{attribute 'no_explicit_call' := 'do not call this POU directly'} 
FUNCTION_BLOCK FB_LoggerProxy IMPLEMENTS I_Logger
VAR_INPUT
END_VAR
VAR_OUTPUT
END_VAR
VAR
	pHead:				POINTER TO ST_LoggerNode;
END_VAR

//FB_Exit muss explizit implementiert werden. Wenn es eine Implementierung gibt, dann wird 
//die Methode aufgerufen, bevor die Steuerung den Code der Funktionsbaustein-Instanz entfernt
//(impliziter Aufruf. Der Rückgabewert wird nicht ausgewertet.
METHOD FB_Exit: BOOL
VAR_INPUT    
bInCopyCode: BOOL;  // TRUE: Die Exit-Methode wird aufgerufen, um die Instanz zu verlassen, die hinterher kopiert wird Online-Change).  
END_VAR
M_Clear();
END_METHOD

METHOD M_Attach : BOOL
VAR_INPUT
    iLogger : I_Logger;
END_VAR
VAR
    pCurrent : POINTER TO ST_LoggerNode;
END_VAR
// invalid input
IF iLogger = 0 THEN
    M_Attach := FALSE;
    RETURN;
END_IF

// first node
IF pHead = 0 THEN
    pHead := __NEW(ST_LoggerNode);
    IF pHead = 0 THEN
        RETURN;
    END_IF
    pHead^.iLogger := iLogger;
    pHead^.pNext := 0;
    M_Attach := TRUE;
    RETURN;
END_IF

// traverse list to check duplicates and reach last node
pCurrent := pHead;
WHILE pCurrent^.pNext <> 0 DO
    IF pCurrent^.iLogger = iLogger THEN
        M_Attach := FALSE; // already attached
        RETURN;
    END_IF
    pCurrent := pCurrent^.pNext;
END_WHILE

// check last node for duplicate
IF pCurrent^.iLogger = iLogger THEN
    RETURN;
END_IF

pCurrent^.pNext:= __NEW(ST_LoggerNode);
IF pCurrent^.pNext = 0 THEN
    RETURN;
END_IF
pCurrent^:= pCurrent^.pNext^;

pCurrent^.iLogger:= iLogger;
pCurrent^.pNext := 0;

M_Attach := TRUE;
END_METHOD

METHOD PUBLIC M_Clear : BOOL
VAR_INPUT
END_VAR
VAR
    pCurrent : POINTER TO ST_LoggerNode;
    pNext    : POINTER TO ST_LoggerNode;
END_VAR
pCurrent := pHead;

WHILE pCurrent <> 0 DO
    pNext := pCurrent^.pNext; // save next pointer
    __DELETE(pCurrent);       // free current node
    pCurrent := pNext;        // move to next node
END_WHILE

pHead := 0;                   // reset head
M_Clear := TRUE;
END_METHOD

METHOD M_Detach : BOOL
VAR_INPUT
	iLogger:			I_Logger;
END_VAR
VAR
    pCurrent : POINTER TO ST_LoggerNode;
    pPrev : POINTER TO ST_LoggerNode;
END_VAR
// invalid input
IF iLogger = 0 THEN
    RETURN;
END_IF

pCurrent := pHead;
pPrev := 0;
WHILE pCurrent <> 0 DO
    IF pCurrent^.iLogger = iLogger THEN
        IF pPrev = 0 THEN
            pHead := pCurrent^.pNext;
        ELSE
            pPrev^.pNext := pCurrent^.pNext;
        END_IF
        __DELETE(pCurrent);
        M_Detach := TRUE;
        RETURN;
    END_IF
    pPrev := pCurrent;
    pCurrent := pCurrent^.pNext;
END_WHILE

M_Detach := FALSE;
END_METHOD

METHOD M_Log : BOOL
VAR_INPUT
	fbMessage	: FB_Message;
END_VAR
VAR
    pCurrent : POINTER TO ST_LoggerNode:= pHead;
END_VAR
WHILE pCurrent <> 0 DO
    pCurrent^.iLogger.M_Log(fbMessage);
    pCurrent := pCurrent^.pNext;
END_WHILE
M_Log := TRUE;
END_METHOD

END_FUNCTION_BLOCK

(* stored: Version 1.1.0.1
   POU FB_LoggerProxy: Id {c92161d9-49ae-4c50-bdac-f079e9b056c0}, SpecialFunc None
   Method FB_Exit: Id {5ffdbfed-bc35-4ea0-a3e2-08b0a045fdd8}
   Method M_Attach: Id {a672c9f6-c6e5-42cc-9e0b-921d3f608c6a}
   Method M_Clear: Id {e2bb2554-8db9-48a3-bb8b-1e817023fd88}
   Method M_Detach: Id {abdf1d3f-b4ea-47b4-a7bf-8742c13025eb}
   Method M_Log: Id {eb21a125-c7d6-460d-84cb-3d1cb4ea2fdf} *)
